PROGRAM ManualVerAxis
VAR
END_VAR

VAVL.axis.ReadStatus();


VAVL.axisPower(
	Axis:= VAVL.axis,
	Enable:= VAVL.enable,
	Enable_Positive:= VAVL.enable,
	Enable_Negative:= VAVL.enable,
	Override:= VAVL.override,
	BufferMode:= ,
	Options:= ,
	Status=> VAVL.running,
	Busy=> ,
	Active=> ,
	Error=> ,
	ErrorID=> VAVL.currentError
);

VAVL.axisMoveManual(
	Axis:= VAVL.axis,
	JogForward:= VAVL.ascend,
	JogBackwards:= VAVL.descend,
	Mode:= ,
	Position:= ,
	Velocity:= ,
	Acceleration:= ,
	Deceleration:= ,
	Jerk:= ,
	Done=> VAVL.done,
	Busy=> VAVL.busy,
	Active=> ,
	CommandAborted=> ,
	Error=> ,
	ErrorID=> VAVL.currentError
);
	
IF VAVL.busy THEN
	VAVL.axisReadActualPosition(Axis := VAVL.axis, Enable := TRUE, Valid=>, Busy=>, Error=>, ErrorID=>, Position=> VAVL.actualPosition);
END_IF
VAVL.actualPositionInt := LREAL_TO_INT(VAVL.actualPosition);

VAVL.axisErrorReset(Axis := VAVL.axis, Execute := VAVL.resetError, Done =>, Error =>, ErrorID => VAVL.currentError);

END_PROGRAM

(* stored: Version 1.1.0.1, ProductVersion 3.1.4024.6
   POU ManualVerAxis: Id {8aa2dc10-decc-4252-95ac-12154723a6ff}, SpecialFunc None *)
